(* IEC 61131-3 sources: ae-debugging/src/funcProgram, 2 files *)

(* ---- func.st ---- *)
NAMESPACE OuterNamespace
    FUNCTION MyFunction : INT
        VAR_INPUT
            in : INT;
        END_VAR
        VAR_OUTPUT
            out : INT;
        END_VAR
        VAR_TEMP
            temp : INT;
        END_VAR
        VAR CONSTANT
            const : INT := 732;
        END_VAR

        temp := in + const;
        temp := temp MOD 10;
        out := temp;
        MyFunction := temp;
    END_FUNCTION
END_NAMESPACE

(* ---- funcProgram.st ---- *)
PROGRAM FuncProgram
    VAR_EXTERNAL
        GlobalInt : INT;
    END_VAR

    VAR
        localInt : INT;
    END_VAR

    GlobalInt := OuterNamespace.MyFunction(GlobalInt, localInt);
END_PROGRAM
